REGION Network 63: UNIT 3 MEASURING PLC PC MINOR VERSIONS MISMATCH WARNING
   RUNG wire#powerrail
      { S7_Templates := "SrcType := UInt" } NE_Contact(in1 := "DB16007_U3_MEAS_STA_MEAS_B_CLIENT_INTERFACE".U03_FACE_B_MEAS_Read.Variable."Version.Minor", in2 := #VERSIONS_MINOR)
      Contact( "DB7259_UNIT_3_STA_MEAS_B_ENABLE_DISABLE".ENABLED )
      wire#w1
      Coil( "DB16000_OPC_UA_TRIGGER_ALARM".CLIENT.U3_MEAS_STA_MEAS_N.ALARMS.PLC_PC_MINOR_VERSIONS_MISMATCH_W )
   END_RUNG
   RUNG wire#w1
      Coil( "DB426_ALARMS_WARNINGS".ALARMS.WARNINGS."742137" )
   END_RUNG
   // the same network as SCL:
   "DB16000_OPC_UA_TRIGGER_ALARM".CLIENT.U3_MEAS_STA_MEAS_N.ALARMS.PLC_PC_MINOR_VERSIONS_MISMATCH_W := ("DB16007_U3_MEAS_STA_MEAS_B_CLIENT_INTERFACE".U03_FACE_B_MEAS_Read.Variable."Version.Minor" <> #VERSIONS_MINOR) AND "DB7259_UNIT_3_STA_MEAS_B_ENABLE_DISABLE".ENABLED;
   "DB426_ALARMS_WARNINGS".ALARMS.WARNINGS."742137" := "DB16000_OPC_UA_TRIGGER_ALARM".CLIENT.U3_MEAS_STA_MEAS_N.ALARMS.PLC_PC_MINOR_VERSIONS_MISMATCH_W;
END_REGION

REGION Network 64: UNIT 3 MEASURING PLC PC MAJOR VERSIONS MISMATCH ALARM
   RUNG wire#powerrail
      { S7_Templates := "SrcType := UInt" } NE_Contact(in1 := "DB16007_U3_MEAS_STA_MEAS_B_CLIENT_INTERFACE".U03_FACE_B_MEAS_Read.Variable."Version.Major", in2 := #VERSIONS_MAJOR)
      wire#w1
      Contact( "DB7259_UNIT_3_STA_MEAS_B_ENABLE_DISABLE".ENABLED )
      wire#w3
      Coil( "DB16000_OPC_UA_TRIGGER_ALARM".CLIENT.U3_MEAS_STA_MEAS_N.ALARMS.PLC_PC_MAJOR_VERSIONS_MISMATCH_A )
   END_RUNG
   RUNG wire#powerrail
      Contact( "DB16000_OPC_UA_TRIGGER_ALARM".CLIENT.U3_MEAS_STA_MEAS_N.ALARMS.PLC_PC_MAJOR_VERSIONS_MISMATCH_A )
      I_Contact( "DB2120_MPP_ITC_IPC".RESET_FAULTS )
      wire#w2
      I_Contact( "DB7300_INTERLOCK_GENERAL".GENERAL_MACHINE.FROM_CELL_TO_MACHINE_GENERAL.MEAS_STA_RESET )
   END_RUNG wire#w1
   RUNG wire#w2
      I_Contact( "DB2001_MODES_GENERAL".MG_AUX_OPTIONS.AUX_BOOL[0] )
   END_RUNG wire#w1
   RUNG wire#w3
      Coil( "DB426_ALARMS_WARNINGS".ALARMS.UNIT_03.FACE_N_MEASURING."724413" )
   END_RUNG
   // the same network as SCL:
   "DB16000_OPC_UA_TRIGGER_ALARM".CLIENT.U3_MEAS_STA_MEAS_N.ALARMS.PLC_PC_MAJOR_VERSIONS_MISMATCH_A := (("DB16007_U3_MEAS_STA_MEAS_B_CLIENT_INTERFACE".U03_FACE_B_MEAS_Read.Variable."Version.Major" <> #VERSIONS_MAJOR) OR ("DB16000_OPC_UA_TRIGGER_ALARM".CLIENT.U3_MEAS_STA_MEAS_N.ALARMS.PLC_PC_MAJOR_VERSIONS_MISMATCH_A AND NOT "DB2120_MPP_ITC_IPC".RESET_FAULTS AND (NOT "DB7300_INTERLOCK_GENERAL".GENERAL_MACHINE.FROM_CELL_TO_MACHINE_GENERAL.MEAS_STA_RESET OR NOT "DB2001_MODES_GENERAL".MG_AUX_OPTIONS.AUX_BOOL[0]))) AND "DB7259_UNIT_3_STA_MEAS_B_ENABLE_DISABLE".ENABLED;
   "DB426_ALARMS_WARNINGS".ALARMS.UNIT_03.FACE_N_MEASURING."724413" := "DB16000_OPC_UA_TRIGGER_ALARM".CLIENT.U3_MEAS_STA_MEAS_N.ALARMS.PLC_PC_MAJOR_VERSIONS_MISMATCH_A;
END_REGION

REGION Network 65: IS_SEOC ALARMS
   RUNG wire#powerrail
      Contact( "M_ONE" )
      wire#w1
      I_Contact( "DB16000_OPC_UA_TRIGGER_ALARM".CLIENT.U3_MEAS_STA_MEAS_N.ALARMS.MEAS_CONNECTION_A )
      I_Contact( "DB16000_OPC_UA_TRIGGER_ALARM".CLIENT.U3_MEAS_STA_MEAS_N.ALARMS.MEAS_METHOD_WORKING_BLOCKED_A )
      I_Contact( "DB16000_OPC_UA_TRIGGER_ALARM".CLIENT.U3_MEAS_STA_MEAS_N.ALARMS.CALIBRATE_CONNECTION_A )
      I_Contact( "DB16000_OPC_UA_TRIGGER_ALARM".CLIENT.U3_MEAS_STA_MEAS_N.ALARMS.CALIBRATE_METHOD_WORKING_BLOCKED_A )
      I_Contact( "DB16000_OPC_UA_TRIGGER_ALARM".CLIENT.U3_MEAS_STA_MEAS_N.ALARMS.RESET_CONNECTION_A )
      I_Contact( "DB16000_OPC_UA_TRIGGER_ALARM".CLIENT.U3_MEAS_STA_MEAS_N.ALARMS.RESET_METHOD_WORKING_BLOCKED_A )
      I_Contact( "DB16000_OPC_UA_TRIGGER_ALARM".CLIENT.U3_MEAS_STA_MEAS_N.ALARMS.READ_VAR_CONNECTION_A )
      I_Contact( "DB16000_OPC_UA_TRIGGER_ALARM".CLIENT.U3_MEAS_STA_MEAS_N.ALARMS.READ_VAR_METHOD_WORKING_BLOCKED_A )
      Not()
      Coil( #AUX_ALARMS )
   END_RUNG
   RUNG wire#w1
      I_Contact( #AUX_ALARMS )
      I_Contact( "DB16000_OPC_UA_TRIGGER_ALARM".CLIENT.U3_MEAS_STA_MEAS_N.ALARMS.PROFILER_CONFIG_A )
      I_Contact( "DB16000_OPC_UA_TRIGGER_ALARM".CLIENT.U3_MEAS_STA_MEAS_N.ALARMS.ANALYZER_CONFIG_A )
      I_Contact( "DB16000_OPC_UA_TRIGGER_ALARM".CLIENT.U3_MEAS_STA_MEAS_N.ALARMS.DMC_STRUCTURE_A )
      I_Contact( "DB16000_OPC_UA_TRIGGER_ALARM".CLIENT.U3_MEAS_STA_MEAS_N.ALARMS.ACQUISITION_A )
      I_Contact( "DB16000_OPC_UA_TRIGGER_ALARM".CLIENT.U3_MEAS_STA_MEAS_N.ALARMS.PROFILER_INIT_A )
      I_Contact( "DB16000_OPC_UA_TRIGGER_ALARM".CLIENT.U3_MEAS_STA_MEAS_N.ALARMS.UMBRELLA_A )
      I_Contact( "DB16000_OPC_UA_TRIGGER_ALARM".CLIENT.U3_MEAS_STA_MEAS_N.ALARMS.RUNOUT_A )
      I_Contact( "DB16000_OPC_UA_TRIGGER_ALARM".CLIENT.U3_MEAS_STA_MEAS_N.ALARMS.DISTANCE_CALCULATION_A )
      I_Contact( "DB16000_OPC_UA_TRIGGER_ALARM".CLIENT.U3_MEAS_STA_MEAS_N.ALARMS.LAYER_GROWTH_A )
      I_Contact( "DB16000_OPC_UA_TRIGGER_ALARM".CLIENT.U3_MEAS_STA_MEAS_N.ALARMS.SURFACE_DEFECTS_A )
      I_Contact( "DB16000_OPC_UA_TRIGGER_ALARM".CLIENT.U3_MEAS_STA_MEAS_N.ALARMS.STORAGE_A )
      I_Contact( "DB16000_OPC_UA_TRIGGER_ALARM".CLIENT.U3_MEAS_STA_MEAS_N.ALARMS.DATABASE_CONNECTION_A )
      I_Contact( "DB16000_OPC_UA_TRIGGER_ALARM".CLIENT.U3_MEAS_STA_MEAS_N.ALARMS.CALIBRATION_MISSING_A )
      I_Contact( "DB16000_OPC_UA_TRIGGER_ALARM".CLIENT.U3_MEAS_STA_MEAS_N.ALARMS.CALIBRATION_PROC_A )
      I_Contact( "DB16000_OPC_UA_TRIGGER_ALARM".CLIENT.U3_MEAS_STA_MEAS_N.ALARMS.PLC_PC_MAJOR_VERSIONS_MISMATCH_A )
      Not()
      Move(in := 16017, out1 => "DB440_MACHINE_ALARM_DECODING".GLOBAL_ALARMS_MACHINE.ALARM_DECODING)
      Contact( "M_DUMMY_OFF" )
      S_Coil( "DB440_MACHINE_ALARM_DECODING".ALARMS_UNIT_3.IS_SEOC_ALARMS )
   END_RUNG
   // the same network as SCL:
   #AUX_ALARMS := NOT ("M_ONE" AND NOT "DB16000_OPC_UA_TRIGGER_ALARM".CLIENT.U3_MEAS_STA_MEAS_N.ALARMS.MEAS_CONNECTION_A AND NOT "DB16000_OPC_UA_TRIGGER_ALARM".CLIENT.U3_MEAS_STA_MEAS_N.ALARMS.MEAS_METHOD_WORKING_BLOCKED_A AND NOT "DB16000_OPC_UA_TRIGGER_ALARM".CLIENT.U3_MEAS_STA_MEAS_N.ALARMS.CALIBRATE_CONNECTION_A AND NOT "DB16000_OPC_UA_TRIGGER_ALARM".CLIENT.U3_MEAS_STA_MEAS_N.ALARMS.CALIBRATE_METHOD_WORKING_BLOCKED_A AND NOT "DB16000_OPC_UA_TRIGGER_ALARM".CLIENT.U3_MEAS_STA_MEAS_N.ALARMS.RESET_CONNECTION_A AND NOT "DB16000_OPC_UA_TRIGGER_ALARM".CLIENT.U3_MEAS_STA_MEAS_N.ALARMS.RESET_METHOD_WORKING_BLOCKED_A AND NOT "DB16000_OPC_UA_TRIGGER_ALARM".CLIENT.U3_MEAS_STA_MEAS_N.ALARMS.READ_VAR_CONNECTION_A AND NOT "DB16000_OPC_UA_TRIGGER_ALARM".CLIENT.U3_MEAS_STA_MEAS_N.ALARMS.READ_VAR_METHOD_WORKING_BLOCKED_A);
   #_w1 := NOT ("M_ONE" AND NOT #AUX_ALARMS AND NOT "DB16000_OPC_UA_TRIGGER_ALARM".CLIENT.U3_MEAS_STA_MEAS_N.ALARMS.PROFILER_CONFIG_A AND NOT "DB16000_OPC_UA_TRIGGER_ALARM".CLIENT.U3_MEAS_STA_MEAS_N.ALARMS.ANALYZER_CONFIG_A AND NOT "DB16000_OPC_UA_TRIGGER_ALARM".CLIENT.U3_MEAS_STA_MEAS_N.ALARMS.DMC_STRUCTURE_A AND NOT "DB16000_OPC_UA_TRIGGER_ALARM".CLIENT.U3_MEAS_STA_MEAS_N.ALARMS.ACQUISITION_A AND NOT "DB16000_OPC_UA_TRIGGER_ALARM".CLIENT.U3_MEAS_STA_MEAS_N.ALARMS.PROFILER_INIT_A AND NOT "DB16000_OPC_UA_TRIGGER_ALARM".CLIENT.U3_MEAS_STA_MEAS_N.ALARMS.UMBRELLA_A AND NOT "DB16000_OPC_UA_TRIGGER_ALARM".CLIENT.U3_MEAS_STA_MEAS_N.ALARMS.RUNOUT_A AND NOT "DB16000_OPC_UA_TRIGGER_ALARM".CLIENT.U3_MEAS_STA_MEAS_N.ALARMS.DISTANCE_CALCULATION_A AND NOT "DB16000_OPC_UA_TRIGGER_ALARM".CLIENT.U3_MEAS_STA_MEAS_N.ALARMS.LAYER_GROWTH_A AND NOT "DB16000_OPC_UA_TRIGGER_ALARM".CLIENT.U3_MEAS_STA_MEAS_N.ALARMS.SURFACE_DEFECTS_A AND NOT "DB16000_OPC_UA_TRIGGER_ALARM".CLIENT.U3_MEAS_STA_MEAS_N.ALARMS.STORAGE_A AND NOT "DB16000_OPC_UA_TRIGGER_ALARM".CLIENT.U3_MEAS_STA_MEAS_N.ALARMS.DATABASE_CONNECTION_A AND NOT "DB16000_OPC_UA_TRIGGER_ALARM".CLIENT.U3_MEAS_STA_MEAS_N.ALARMS.CALIBRATION_MISSING_A AND NOT "DB16000_OPC_UA_TRIGGER_ALARM".CLIENT.U3_MEAS_STA_MEAS_N.ALARMS.CALIBRATION_PROC_A AND NOT "DB16000_OPC_UA_TRIGGER_ALARM".CLIENT.U3_MEAS_STA_MEAS_N.ALARMS.PLC_PC_MAJOR_VERSIONS_MISMATCH_A);
   IF #_w1 THEN "DB440_MACHINE_ALARM_DECODING".GLOBAL_ALARMS_MACHINE.ALARM_DECODING := 16017; END_IF;
   IF #_w1 AND "M_DUMMY_OFF" THEN
       "DB440_MACHINE_ALARM_DECODING".ALARMS_UNIT_3.IS_SEOC_ALARMS := TRUE;
   END_IF;
END_REGION

REGION Network 66: SEOC ALARMS
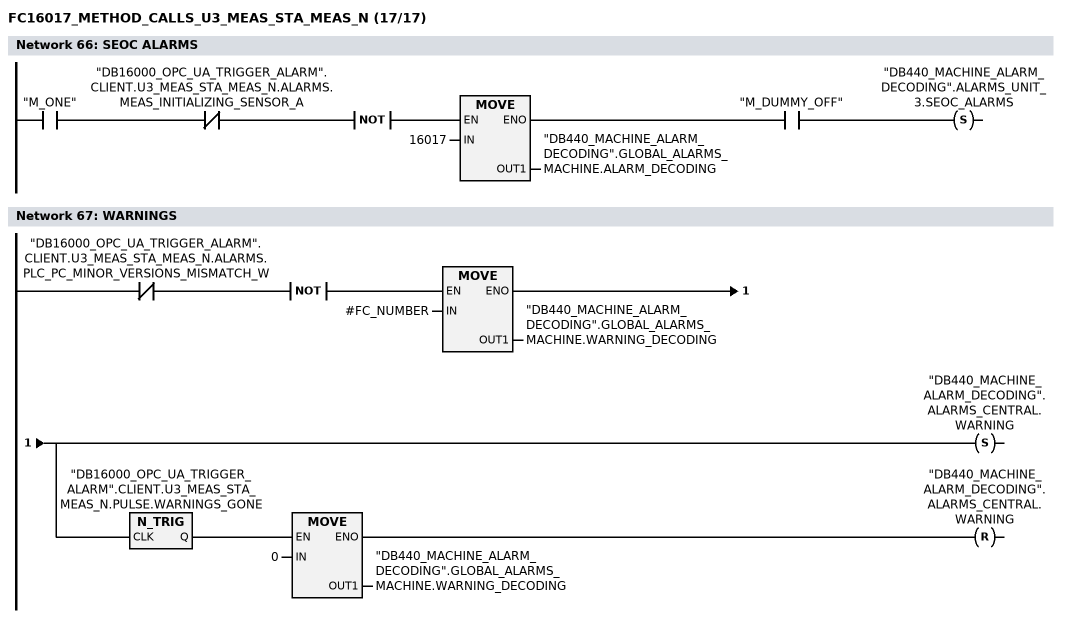
   RUNG wire#powerrail
      Contact( "M_ONE" )
      I_Contact( "DB16000_OPC_UA_TRIGGER_ALARM".CLIENT.U3_MEAS_STA_MEAS_N.ALARMS.MEAS_INITIALIZING_SENSOR_A )
      Not()
      Move(in := 16017, out1 => "DB440_MACHINE_ALARM_DECODING".GLOBAL_ALARMS_MACHINE.ALARM_DECODING)
      Contact( "M_DUMMY_OFF" )
      S_Coil( "DB440_MACHINE_ALARM_DECODING".ALARMS_UNIT_3.SEOC_ALARMS )
   END_RUNG
   // the same network as SCL:
   #_w1 := NOT ("M_ONE" AND NOT "DB16000_OPC_UA_TRIGGER_ALARM".CLIENT.U3_MEAS_STA_MEAS_N.ALARMS.MEAS_INITIALIZING_SENSOR_A);
   IF #_w1 THEN "DB440_MACHINE_ALARM_DECODING".GLOBAL_ALARMS_MACHINE.ALARM_DECODING := 16017; END_IF;
   IF #_w1 AND "M_DUMMY_OFF" THEN "DB440_MACHINE_ALARM_DECODING".ALARMS_UNIT_3.SEOC_ALARMS := TRUE; END_IF;
END_REGION

REGION Network 67: WARNINGS
   RUNG wire#powerrail
      I_Contact( "DB16000_OPC_UA_TRIGGER_ALARM".CLIENT.U3_MEAS_STA_MEAS_N.ALARMS.PLC_PC_MINOR_VERSIONS_MISMATCH_W )
      Not()
      Move(in := #FC_NUMBER, out1 => "DB440_MACHINE_ALARM_DECODING".GLOBAL_ALARMS_MACHINE.WARNING_DECODING)
      wire#w1
      S_Coil( "DB440_MACHINE_ALARM_DECODING".ALARMS_CENTRAL.WARNING )
   END_RUNG
   RUNG wire#w1
      N_Trig( "DB16000_OPC_UA_TRIGGER_ALARM".CLIENT.U3_MEAS_STA_MEAS_N.PULSE.WARNINGS_GONE )
      Move(in := 0, out1 => "DB440_MACHINE_ALARM_DECODING".GLOBAL_ALARMS_MACHINE.WARNING_DECODING)
      R_Coil( "DB440_MACHINE_ALARM_DECODING".ALARMS_CENTRAL.WARNING )
   END_RUNG
   // the same network as SCL:
   #_w1 := NOT (NOT "DB16000_OPC_UA_TRIGGER_ALARM".CLIENT.U3_MEAS_STA_MEAS_N.ALARMS.PLC_PC_MINOR_VERSIONS_MISMATCH_W);
   IF #_w1 THEN
       "DB440_MACHINE_ALARM_DECODING".GLOBAL_ALARMS_MACHINE.WARNING_DECODING := #FC_NUMBER;
       "DB440_MACHINE_ALARM_DECODING".ALARMS_CENTRAL.WARNING := TRUE;
   END_IF;
   #_w2 := NOT #_w1 AND "DB16000_OPC_UA_TRIGGER_ALARM".CLIENT.U3_MEAS_STA_MEAS_N.PULSE.WARNINGS_GONE;   // falling edge
   "DB16000_OPC_UA_TRIGGER_ALARM".CLIENT.U3_MEAS_STA_MEAS_N.PULSE.WARNINGS_GONE := #_w1;
   IF #_w2 THEN
       "DB440_MACHINE_ALARM_DECODING".GLOBAL_ALARMS_MACHINE.WARNING_DECODING := 0;
       "DB440_MACHINE_ALARM_DECODING".ALARMS_CENTRAL.WARNING := FALSE;
   END_IF;
END_REGION
END_FUNCTION
